PROGRAM Light 
VAR
	output2 : BOOL;
	input2 : BOOL;
END_VAR

output2 := input2;

END_PROGRAM

(* stored: Version 1.1.0.1, ProductVersion 3.1.4024.12
   POU Light: Id {690aaac3-e251-4371-964b-125c2906d72d}, SpecialFunc None *)
